{attribute 'TcDependOnClassFactory' := 'WeldingArm6AxisMotion_Control'}
FUNCTION_BLOCK FB_WeldingArm6AxisMotion_Control EXTENDS FB_TcMatSimObject
VAR_INPUT
	stInput: ST_WeldingArm6AxisMotion_Control_Input;
END_VAR
VAR_OUTPUT
	stOutput: ST_WeldingArm6AxisMotion_Control_Output;
END_VAR
VAR
	stInitData: ST_WeldingArm6AxisMotion_Control_InitData;
	arrDataAreas: ARRAY[1..2] OF ST_TcMatSimObjectDataAreaInfo;
	bParametersVerified: BOOL;
END_VAR

PROPERTY CallBy_Online : TctModuleCallByType
GET
hResult := GetObjPara(16#00000000,sizeof(CallBy_Online),adr(CallBy_Online));
END_GET
SET
hResult := SetObjPara(16#00000000,sizeof(CallBy_Online),adr(CallBy_Online));
END_SET
END_PROPERTY

PROPERTY CallBy_Startup : TctModuleCallByType
GET
CallBy_Startup := stInitData.CallBy;
END_GET
SET
stInitData.CallBy := CallBy_Startup;
END_SET
END_PROPERTY

PROPERTY ContextInfoArr_0_TaskCycleTimeNs_Online : UDINT
GET
hResult := GetObjPara(16#03002080,sizeof(ContextInfoArr_0_TaskCycleTimeNs_Online),adr(ContextInfoArr_0_TaskCycleTimeNs_Online));
END_GET
SET
hResult := SetObjPara(16#03002080,sizeof(ContextInfoArr_0_TaskCycleTimeNs_Online),adr(ContextInfoArr_0_TaskCycleTimeNs_Online));
END_SET
END_PROPERTY

PROPERTY ContextInfoArr_0_TaskCycleTimeNs_Startup : UDINT
GET
ContextInfoArr_0_TaskCycleTimeNs_Startup := stInitData.ContextInfoArr_0_TaskCycleTimeNs;
END_GET
SET
stInitData.ContextInfoArr_0_TaskCycleTimeNs := ContextInfoArr_0_TaskCycleTimeNs_Startup;
END_SET
END_PROPERTY

PROPERTY ContextInfoArr_0_TaskOid_Online : OTCID
GET
hResult := GetObjPara(16#03002060,sizeof(ContextInfoArr_0_TaskOid_Online),adr(ContextInfoArr_0_TaskOid_Online));
END_GET
SET
hResult := SetObjPara(16#03002060,sizeof(ContextInfoArr_0_TaskOid_Online),adr(ContextInfoArr_0_TaskOid_Online));
END_SET
END_PROPERTY

PROPERTY ContextInfoArr_0_TaskOid_Startup : OTCID
GET
ContextInfoArr_0_TaskOid_Startup := stInitData.ContextInfoArr_0_TaskOid;
END_GET
SET
stInitData.ContextInfoArr_0_TaskOid := ContextInfoArr_0_TaskOid_Startup;
END_SET
END_PROPERTY

PROPERTY ContextInfoArr_0_TaskPort_Online : UINT
GET
hResult := GetObjPara(16#03002090,sizeof(ContextInfoArr_0_TaskPort_Online),adr(ContextInfoArr_0_TaskPort_Online));
END_GET
SET
hResult := SetObjPara(16#03002090,sizeof(ContextInfoArr_0_TaskPort_Online),adr(ContextInfoArr_0_TaskPort_Online));
END_SET
END_PROPERTY

PROPERTY ContextInfoArr_0_TaskPort_Startup : UINT
GET
ContextInfoArr_0_TaskPort_Startup := stInitData.ContextInfoArr_0_TaskPort;
END_GET
SET
stInitData.ContextInfoArr_0_TaskPort := ContextInfoArr_0_TaskPort_Startup;
END_SET
END_PROPERTY

PROPERTY ContextInfoArr_0_TaskPriority_Online : UDINT
GET
hResult := GetObjPara(16#03002070,sizeof(ContextInfoArr_0_TaskPriority_Online),adr(ContextInfoArr_0_TaskPriority_Online));
END_GET
SET
hResult := SetObjPara(16#03002070,sizeof(ContextInfoArr_0_TaskPriority_Online),adr(ContextInfoArr_0_TaskPriority_Online));
END_SET
END_PROPERTY

PROPERTY ContextInfoArr_0_TaskPriority_Startup : UDINT
GET
ContextInfoArr_0_TaskPriority_Startup := stInitData.ContextInfoArr_0_TaskPriority;
END_GET
SET
stInitData.ContextInfoArr_0_TaskPriority := ContextInfoArr_0_TaskPriority_Startup;
END_SET
END_PROPERTY

PROPERTY ContextInfoArr_0_TaskSortOrder_Online : UDINT
GET
hResult := GetObjPara(16#030020b0,sizeof(ContextInfoArr_0_TaskSortOrder_Online),adr(ContextInfoArr_0_TaskSortOrder_Online));
END_GET
SET
hResult := SetObjPara(16#030020b0,sizeof(ContextInfoArr_0_TaskSortOrder_Online),adr(ContextInfoArr_0_TaskSortOrder_Online));
END_SET
END_PROPERTY

PROPERTY ContextInfoArr_0_TaskSortOrder_Startup : UDINT
GET
ContextInfoArr_0_TaskSortOrder_Startup := stInitData.ContextInfoArr_0_TaskSortOrder;
END_GET
SET
stInitData.ContextInfoArr_0_TaskSortOrder := ContextInfoArr_0_TaskSortOrder_Startup;
END_SET
END_PROPERTY

PROPERTY CycleUpdateExecuted_Online : BOOL
GET
hResult := GetObjPara(16#00000004,sizeof(CycleUpdateExecuted_Online),adr(CycleUpdateExecuted_Online));
END_GET
SET
hResult := SetObjPara(16#00000004,sizeof(CycleUpdateExecuted_Online),adr(CycleUpdateExecuted_Online));
END_SET
END_PROPERTY

METHOD Execute : HRESULT

IF (SUCCEEDED(hResult)) THEN
  hResult := VerifyParameters();
END_IF

	// update DataArea information
SetDataAreaInfo(ADR(arrDataAreas),2);
	
	// call base method
Execute := SUPER^.Execute();
END_METHOD

PROPERTY ExecuteModelCode_Online : BOOL
GET
hResult := GetObjPara(16#00000008,sizeof(ExecuteModelCode_Online),adr(ExecuteModelCode_Online));
END_GET
SET
hResult := SetObjPara(16#00000008,sizeof(ExecuteModelCode_Online),adr(ExecuteModelCode_Online));
END_SET
END_PROPERTY

PROPERTY ExecuteModelCode_Startup : BOOL
GET
ExecuteModelCode_Startup := stInitData.ExecuteModelCode;
END_GET
SET
stInitData.ExecuteModelCode := ExecuteModelCode_Startup;
END_SET
END_PROPERTY

PROPERTY ExecutionSequence_Online : TctModuleExecutionSequenceType
GET
hResult := GetObjPara(16#00000001,sizeof(ExecutionSequence_Online),adr(ExecutionSequence_Online));
END_GET
SET
hResult := SetObjPara(16#00000001,sizeof(ExecutionSequence_Online),adr(ExecutionSequence_Online));
END_SET
END_PROPERTY

PROPERTY ExecutionSequence_Startup : TctModuleExecutionSequenceType
GET
ExecutionSequence_Startup := stInitData.ExecutionSequence;
END_GET
SET
stInitData.ExecutionSequence := ExecutionSequence_Startup;
END_SET
END_PROPERTY

METHOD FB_init : BOOL
VAR_INPUT
	/// if TRUE, the retain variables are initialized (warm start / cold start)
	bInitRetains: BOOL;
	/// if TRUE, the instance afterwards gets moved into the copy code (online change)
	bInCopyCode: BOOL;
	oid: OTCID;
END_VAR
VAR
	clsId: CLSID;
END_VAR

// initialize flags
bParametersVerified := false;
                    
// set module class id for compatibility check
clsId.Data1 := 16#412caec1;
clsId.Data2 := 16#7008;
clsId.Data3 := 16#47ed;
clsId.Data4[0] := 16#9b;
clsId.Data4[1] := 16#82;
clsId.Data4[2] := 16#ce;
clsId.Data4[3] := 16#15;
clsId.Data4[4] := 16#e3;
clsId.Data4[5] := 16#d3;
clsId.Data4[6] := 16#23;
clsId.Data4[7] := 16#f9;

AssignClassId(clsId);
                    
// initialize InitData structure with default values              
stInitData.CallByHdr.indexGroup := 0;
stInitData.CallByHdr.indexOffset := 16#00000000;
stInitData.CallByHdr.cbData := SIZEOF(stInitData.CallBy);
stInitData.CallBy := TctModuleCallByType.Module;
stInitData.ExecutionSequenceHdr.indexGroup := 0;
stInitData.ExecutionSequenceHdr.indexOffset := 16#00000001;
stInitData.ExecutionSequenceHdr.cbData := SIZEOF(stInitData.ExecutionSequence);
stInitData.ExecutionSequence := TctModuleExecutionSequenceType.StateUpdateAfterOutputMapping;
stInitData.StepSizeHdr.indexGroup := 0;
stInitData.StepSizeHdr.indexOffset := 16#00000002;
stInitData.StepSizeHdr.cbData := SIZEOF(stInitData.StepSize);
stInitData.StepSize := TctStepSizeType.UseTaskCycleTime;
stInitData.ExecuteModelCodeHdr.indexGroup := 0;
stInitData.ExecuteModelCodeHdr.indexOffset := 16#00000008;
stInitData.ExecuteModelCodeHdr.cbData := SIZEOF(stInitData.ExecuteModelCode);
stInitData.ExecuteModelCode := 1;
stInitData.ModelParametersHdr.indexGroup := 0;
stInitData.ModelParametersHdr.indexOffset := 16#82000000;
stInitData.ModelParametersHdr.cbData := SIZEOF(stInitData.ModelParameters);
stInitData.ModelParameters.tcycle_Value := 5.00000000000000000e+00;
stInitData.ModelParameters.J1rg_Value[0] := 2.00000000000000000e+01;
stInitData.ModelParameters.J1rg_Value[1] := 2.00000000000000000e+02;
stInitData.ModelParameters.J2rg_Value[0] := -2.70000000000000000e+02;
stInitData.ModelParameters.J2rg_Value[1] := 9.00000000000000000e+01;
stInitData.ModelParameters.J3rg_Value[0] := 2.00000000000000000e+01;
stInitData.ModelParameters.J3rg_Value[1] := 1.30000000000000000e+02;
stInitData.ModelParameters.phirg_Value[0] := -3.00000000000000000e+01;
stInitData.ModelParameters.phirg_Value[1] := 3.00000000000000000e+01;
stInitData.ModelParameters.gamarg_Value[0] := 1.50000000000000000e+01;
stInitData.ModelParameters.gamarg_Value[1] := 3.50000000000000000e+01;
stInitData.ContextInfoArr_0_TaskOidHdr.indexGroup := 0;
stInitData.ContextInfoArr_0_TaskOidHdr.indexOffset := 16#03002060;
stInitData.ContextInfoArr_0_TaskOidHdr.cbData := SIZEOF(stInitData.ContextInfoArr_0_TaskOid);
stInitData.ContextInfoArr_0_TaskPriorityHdr.indexGroup := 0;
stInitData.ContextInfoArr_0_TaskPriorityHdr.indexOffset := 16#03002070;
stInitData.ContextInfoArr_0_TaskPriorityHdr.cbData := SIZEOF(stInitData.ContextInfoArr_0_TaskPriority);
stInitData.ContextInfoArr_0_TaskCycleTimeNsHdr.indexGroup := 0;
stInitData.ContextInfoArr_0_TaskCycleTimeNsHdr.indexOffset := 16#03002080;
stInitData.ContextInfoArr_0_TaskCycleTimeNsHdr.cbData := SIZEOF(stInitData.ContextInfoArr_0_TaskCycleTimeNs);
stInitData.ContextInfoArr_0_TaskPortHdr.indexGroup := 0;
stInitData.ContextInfoArr_0_TaskPortHdr.indexOffset := 16#03002090;
stInitData.ContextInfoArr_0_TaskPortHdr.cbData := SIZEOF(stInitData.ContextInfoArr_0_TaskPort);
stInitData.ContextInfoArr_0_TaskSortOrderHdr.indexGroup := 0;
stInitData.ContextInfoArr_0_TaskSortOrderHdr.indexOffset := 16#030020b0;
stInitData.ContextInfoArr_0_TaskSortOrderHdr.cbData := SIZEOF(stInitData.ContextInfoArr_0_TaskSortOrder);
stInitData.Header.cbData := SIZEOF(stInitData)-SIZEOF(stInitData.Header);
stInitData.Header.uiElmCnt := 10;


// set pointer to InitData structure
SetInitDataInfo(ADR(stInitData));

// set DataArea information
SetDataAreaInfo(ADR(arrDataAreas),2);
arrDataAreas[1].nDataAreaId := 0;
arrDataAreas[1].nSize := SIZEOF(stInput);
arrDataAreas[1].pPlcVar := ADR(stInput);
arrDataAreas[1].pModuleProcImg := 0;
arrDataAreas[1].eDataAreaType := E_TcMatSimDataAreaType.InputDst;
arrDataAreas[2].nDataAreaId := 1;
arrDataAreas[2].nSize := SIZEOF(stOutput);
arrDataAreas[2].pPlcVar := ADR(stOutput);
arrDataAreas[2].pModuleProcImg := 0;
arrDataAreas[2].eDataAreaType := E_TcMatSimDataAreaType.OutputSrc;


// initialize basic interface pointers and return
FB_init := SUCCEEDED(Init(oid));
END_METHOD

PROPERTY InitData : ST_WeldingArm6AxisMotion_Control_InitData
GET
InitData := stInitData;
END_GET
SET
stInitData := InitData;
END_SET
END_PROPERTY

PROPERTY Input_Online : ExtU_weldingArm6axisMotionTes_T
GET
hResult := GetObjPara(16#80000000,sizeof(Input_Online),adr(Input_Online));
END_GET
SET
hResult := SetObjPara(16#80000000,sizeof(Input_Online),adr(Input_Online));
END_SET
END_PROPERTY

{attribute 'object_name' := 'Internal_SetObjState'}
METHOD PROTECTED Internal_SetObjState
VAR_INPUT
	hr: REFERENCE TO HRESULT;
	nextState: TCOM_STATE;
END_VAR

// update pointer to InitData structure
SetInitDataInfo(ADR(stInitData));
// call base method
SUPER^.Internal_SetObjState(hr,nextState);
END_METHOD

PROPERTY MdlInitialized_Online : BOOL
GET
hResult := GetObjPara(16#00000003,sizeof(MdlInitialized_Online),adr(MdlInitialized_Online));
END_GET
SET
hResult := SetObjPara(16#00000003,sizeof(MdlInitialized_Online),adr(MdlInitialized_Online));
END_SET
END_PROPERTY

PROPERTY ModelParameters_Online : P_weldingArm6axisMotionTest1_T
GET
hResult := GetObjPara(16#82000000,sizeof(ModelParameters_Online),adr(ModelParameters_Online));
END_GET
SET
hResult := SetObjPara(16#82000000,sizeof(ModelParameters_Online),adr(ModelParameters_Online));
END_SET
END_PROPERTY

PROPERTY ModelParameters_Startup : P_weldingArm6axisMotionTest1_T
GET
ModelParameters_Startup := stInitData.ModelParameters;
END_GET
SET
stInitData.ModelParameters := ModelParameters_Startup;
END_SET
END_PROPERTY

PROPERTY ModuleBuildInfo_Online : TctModuleBuildInfoType
GET
hResult := GetObjPara(16#00000007,sizeof(ModuleBuildInfo_Online),adr(ModuleBuildInfo_Online));
END_GET
SET
hResult := SetObjPara(16#00000007,sizeof(ModuleBuildInfo_Online),adr(ModuleBuildInfo_Online));
END_SET
END_PROPERTY

PROPERTY ModuleInfo_Online : TctModuleInfoType
GET
hResult := GetObjPara(16#00000006,sizeof(ModuleInfo_Online),adr(ModuleInfo_Online));
END_GET
SET
hResult := SetObjPara(16#00000006,sizeof(ModuleInfo_Online),adr(ModuleInfo_Online));
END_SET
END_PROPERTY

{attribute 'object_name' := 'SaveOnlineParametersForInit'}
METHOD SaveOnlineParametersForInit : HRESULT
VAR
	idx: UINT;
	pInitElemHdr: POINTER TO TComInitDataElmHdr;
	pData: PVOID;
	nData: UDINT;
END_VAR
VAR CONSTANT
	nInitDataAlignment: UDINT := 4;
END_VAR

// update pointer to InitData structure
SetInitDataInfo(ADR(stInitData));
// call base method
SaveOnlineParametersForInit := SUPER^.SaveOnlineParametersForInit();
END_METHOD

PROPERTY SimulinkTime_Online : LREAL
GET
hResult := GetObjPara(16#00000005,sizeof(SimulinkTime_Online),adr(SimulinkTime_Online));
END_GET
SET
hResult := SetObjPara(16#00000005,sizeof(SimulinkTime_Online),adr(SimulinkTime_Online));
END_SET
END_PROPERTY

PROPERTY StepSize_Online : TctStepSizeType
GET
hResult := GetObjPara(16#00000002,sizeof(StepSize_Online),adr(StepSize_Online));
END_GET
SET
hResult := SetObjPara(16#00000002,sizeof(StepSize_Online),adr(StepSize_Online));
END_SET
END_PROPERTY

PROPERTY StepSize_Startup : TctStepSizeType
GET
StepSize_Startup := stInitData.StepSize;
END_GET
SET
stInitData.StepSize := StepSize_Startup;
END_SET
END_PROPERTY

{attribute 'object_name' := 'VerifyParameters'}
METHOD PRIVATE VerifyParameters : HRESULT
VAR
	moduleCallByParam: TctModuleCallByType;
END_VAR

IF (bParametersVerified) THEN
  VerifyParameters := Tc2_System.E_HRESULTAdsErr.HRESULT_ADS_NOERROR;
ELSE
  VerifyParameters := GetObjPara(stInitData.CallByHdr.indexOffset,SIZEOF(moduleCallByParam),ADR(moduleCallByParam));
  
  // check the "CallBy" parameter to be set to "Module"
  IF (SUCCEEDED(VerifyParameters) AND (moduleCallByParam <> TctModuleCallByType.Module)) THEN
      VerifyParameters := Tc2_System.E_HRESULTAdsErr.INVALIDPARM;
  END_IF
  
  // set the parameters verified flag
  bParametersVerified := SUCCEEDED(VerifyParameters);
END_IF
END_METHOD

END_FUNCTION_BLOCK

(* stored: Version 1.1.0.1, ProductVersion 3.1.4020.12
   POU FB_WeldingArm6AxisMotion_Control: Id {2a1f7bf2-a416-47b2-b7ce-38d5a19dee8a}, SpecialFunc None
   Property CallBy_Online: Id {348a1fc9-b7bc-46f3-ab96-abdde30b319a}
   Get Get: Id {24849bbd-35f9-4030-a879-5aa74d1da3c3}
   Set Set: Id {cfc95f9d-26e7-4f72-ae82-30a324f2fb89}
   Property CallBy_Startup: Id {209b2854-2b9c-4aa4-9a31-396dbaf87083}
   Get Get: Id {475458a0-bc80-449d-bc5a-0d8bd15db468}
   Set Set: Id {5a348fbd-62ee-4188-845d-2a389605dce7}
   Property ContextInfoArr_0_TaskCycleTimeNs_Online: Id {f57610f1-7966-4765-a49f-ab04507eb225}
   Get Get: Id {9015a13d-809e-4c8b-bf96-9b97d0f57bf5}
   Set Set: Id {c1f6ae2b-a8bc-4d4d-b8f3-acd9741009fe}
   Property ContextInfoArr_0_TaskCycleTimeNs_Startup: Id {24766200-cffe-4d66-b90d-db2396738476}
   Get Get: Id {9a7cce48-9c00-4e03-9bc8-74ecb2d8a96b}
   Set Set: Id {cdb830f8-425e-4d42-a710-92e3c67bfb18}
   Property ContextInfoArr_0_TaskOid_Online: Id {6fe7bb65-bc41-4b43-ac4f-3ba8a5bdc08c}
   Get Get: Id {d8d7e3f0-2ae1-437a-8c1d-ce742c814b4a}
   Set Set: Id {aad0f2b0-3524-45f6-83ec-0a1e1b4db9ff}
   Property ContextInfoArr_0_TaskOid_Startup: Id {93e9fd10-4482-476f-95cf-54520f395618}
   Get Get: Id {7f791cb1-7363-4c5f-9f20-23234b199874}
   Set Set: Id {76f57484-c9cb-4753-87e3-57f4cae1fca9}
   Property ContextInfoArr_0_TaskPort_Online: Id {6328e1ee-38d9-4703-b268-3f8ca8a03a14}
   Get Get: Id {60fca8d8-6298-46f6-a85d-46ad758050a8}
   Set Set: Id {0ba2f6f1-7f54-4baa-be02-78ea2acd65e1}
   Property ContextInfoArr_0_TaskPort_Startup: Id {c01692a5-2dd8-4068-92f0-7f69535bee20}
   Get Get: Id {81963410-94e8-45f9-aaa5-7d221655dc3a}
   Set Set: Id {17404948-cfb5-4eba-9dae-14e6be52121c}
   Property ContextInfoArr_0_TaskPriority_Online: Id {4278e937-76ee-43e3-a03a-1bbe7e610f02}
   Get Get: Id {27a4be9c-5597-4dd4-b7ef-2b55f91584f4}
   Set Set: Id {0b96c88f-7c21-4f6b-a84f-065c9012c0f3}
   Property ContextInfoArr_0_TaskPriority_Startup: Id {c2a7e9be-d9a3-48df-b0ee-bfa54738e810}
   Get Get: Id {86327e1e-8603-47c0-a2b9-02067419ad25}
   Set Set: Id {04f050bf-d54d-440a-bdaa-da84f09a18d6}
   Property ContextInfoArr_0_TaskSortOrder_Online: Id {b6171bff-8bc0-4db0-931b-f266891681d5}
   Get Get: Id {e763cc47-c1d0-43f3-a3b1-8dfeaead0a12}
   Set Set: Id {c79b9351-754e-4ef1-9601-98858ef908cc}
   Property ContextInfoArr_0_TaskSortOrder_Startup: Id {2705c061-8bd7-4fc8-82eb-baa5567d9fa9}
   Get Get: Id {18b7e25b-dc74-4d95-985d-66e892019c06}
   Set Set: Id {64f3233d-98d8-4b88-bdd4-1a8b81c99ef5}
   Property CycleUpdateExecuted_Online: Id {11c0820a-6f74-4d38-a01e-e3d8bcffdeb0}
   Get Get: Id {54634eb9-720d-4bad-bb78-4ef990e2b867}
   Set Set: Id {65169889-1ff9-4420-abc6-09b224dd6ade}
   Method Execute: Id {fb21360d-07a2-4ab9-835d-6778ebe3dcd5}
   Property ExecuteModelCode_Online: Id {32949c4d-5727-4a0d-bb90-9639c9ce3e1a}
   Get Get: Id {e4cd009b-b5a5-4a5c-9fd0-11835f720632}
   Set Set: Id {1715d646-927d-4628-9594-122b753b6408}
   Property ExecuteModelCode_Startup: Id {cf33e0f7-a1d0-4870-ba10-6e4229c5438c}
   Get Get: Id {57588e75-298e-497b-8402-c38d51ff3bcc}
   Set Set: Id {820f65d1-1856-4f4f-9739-d385b15e03f3}
   Property ExecutionSequence_Online: Id {ac733a2c-15b1-4602-b191-6e9a9746b7f9}
   Get Get: Id {18534b8c-c9d6-4efa-8cb0-5bb364f82e36}
   Set Set: Id {663c9a82-85c2-4433-b956-b26eb10c5ab5}
   Property ExecutionSequence_Startup: Id {dd5cbb5e-b6bd-416f-99b7-c714f5fdd4f6}
   Get Get: Id {748269d1-49a5-4cf6-b78e-934de099f857}
   Set Set: Id {fb03f4a1-2857-42bf-8dde-971def52a56e}
   Method FB_init: Id {ba00e333-2925-4114-8af9-f4a1440819f3}
   Property InitData: Id {5473cc14-1bb6-4614-a37b-4ef9ed908a7e}
   Get Get: Id {f8ea60c5-16f3-4e23-89c0-1c7bf81cf9d8}
   Set Set: Id {f4b386d7-26aa-4a5e-bbbd-b919f45f2627}
   Property Input_Online: Id {6ae801c5-7dbe-4c17-83b1-9e2659213e9d}
   Get Get: Id {6409c409-bb54-49bf-a6a5-16d701c5d661}
   Set Set: Id {f9bc47d3-a08b-4d79-8742-afd28c0d2ca6}
   Method Internal_SetObjState: Id {486f4937-6fbf-46d6-8a87-ca0adaf76150}
   Property MdlInitialized_Online: Id {8cde9dfe-669e-4603-b138-b86a036415c1}
   Get Get: Id {941b7d1c-b749-411d-bba8-53050efd64af}
   Set Set: Id {e660b80b-616d-4313-8caa-e11c755acd84}
   Property ModelParameters_Online: Id {7ac5d1eb-0bb1-419c-a226-97bd04122bb0}
   Get Get: Id {ba69a436-53d1-4e61-8126-a87286a561ea}
   Set Set: Id {718274a2-2a87-4ff9-a253-52ea7b34eddc}
   Property ModelParameters_Startup: Id {e11d34d3-f545-4a02-9fe9-10da1f745e16}
   Get Get: Id {9a439858-7e92-456f-a00f-0da18c86e54c}
   Set Set: Id {1dcd4052-1a29-46eb-bfdb-30a60b3beae5}
   Property ModuleBuildInfo_Online: Id {8cdee088-ed87-4235-91bf-d3276b3b5e15}
   Get Get: Id {1462d9da-e674-4223-90db-8faf5f3c7c8b}
   Set Set: Id {6a7cf3fd-bdf6-455a-96df-cbc364134866}
   Property ModuleInfo_Online: Id {f9375b7c-bd9c-457b-9f91-131d96f4260f}
   Get Get: Id {f306f688-b38c-4f92-a0a5-7b0f9bee416c}
   Set Set: Id {caf07d42-839e-474d-900e-4a811dceaee0}
   Method SaveOnlineParametersForInit: Id {689315f5-cfa3-4656-a203-ad0cbf904882}
   Property SimulinkTime_Online: Id {b1bd0378-2c9b-4d27-8b9f-37174419c174}
   Get Get: Id {045d379a-629a-4327-a30f-5d9826fbf0c6}
   Set Set: Id {3e527776-c8e8-4db0-97bb-6ac70170752c}
   Property StepSize_Online: Id {1cbe52d6-bbac-44f5-bd12-811998f7aa78}
   Get Get: Id {f0b7a9a0-fd59-471e-802e-92eda03c9d4b}
   Set Set: Id {f94c98f7-2ba7-43a5-8703-a648f1a52d21}
   Property StepSize_Startup: Id {10fed9f5-abe4-43c2-b948-c9b90907fd57}
   Get Get: Id {557fbd16-ae94-4fba-bc43-24f401e3a963}
   Set Set: Id {7fa9b599-da3e-4f80-8236-4714e30472c8}
   Method VerifyParameters: Id {7c7ba7c2-a467-4051-8eaa-51c629d9ec1d} *)
